TYPE ST_ModuleCmd :
STRUCT
END_STRUCT
END_TYPE

(* stored: Version 1.1.0.1, ProductVersion 3.1.4026.17
   DUT ST_ModuleCmd: Id {305cc7b5-54f9-4cfa-ace0-763be832c127} *)
